FUNCTION_BLOCK FB_Basisfunktionalitaeten
VAR_INPUT
END_VAR
VAR_OUTPUT
END_VAR
VAR
	V_Start			:BOOL;		// Variable für internes handling der Eigenschaft 
	V_Stop			:BOOL;		// Variable für internes handling der Eigenschaft 
END_VAR

METHOD M_START : BOOL
VAR_INPUT
END_VAR
V_Start := 1;
V_Stop := 0;
END_METHOD

METHOD M_STOP : BOOL
VAR_INPUT
END_VAR
V_Start := 0;
V_Stop := 1;
END_METHOD

PROPERTY P_Ready : BOOL
GET
P_Ready := V_Stop;
END_GET
END_PROPERTY

END_FUNCTION_BLOCK

(* stored: Version 1.1.0.1, ProductVersion 3.1.4024.12
   POU FB_Basisfunktionalitaeten: Id {fffd0907-c1c1-493c-ac2c-314e9089ee0d}, SpecialFunc None
   Method M_START: Id {814a3d4c-bdf1-4ff2-b4ec-cf40aba645ba}
   Method M_STOP: Id {645c63c8-13f0-478f-ae7b-32e8477e4722}
   Property P_Ready: Id {ffbbd73b-900a-4aee-bc8d-5f319a8cfba9}
   Get Get: Id {7a5f06a2-1350-4bac-a53f-e294f574a899} *)
